//==================================================================================================
//							Beckhoff Automation Poland
//									18.04.2018
//	Struktura zawierajaca I/O odpowiedniego bloku
//  v1.0	|| TC v 3.1.4022.16		|| - pierwsza wersja
//==================================================================================================
TYPE ST_MCPowerIO:
STRUCT
	bEnable							: BOOL;
	bEnable_Positive				: BOOL;
	bEnable_Negative				: BOOL;
	lrOverride						: LREAL := 100.0;
	eBufferMode						: Tc2_MC2.MC_BufferMode;
	stOptions						: Tc2_MC2.ST_PowerOptions;
	bStatus							: bool; // Same meaning as Done
	bBusy							: BOOL;
	bActive							: BOOL;
	bError							: BOOL;
	udiErrorID						: UDINT;
END_STRUCT
END_TYPE

(* stored: Version 1.1.0.1, ProductVersion 3.1.4026.13, FileIdentifier 2b62fc5234dd54785e8d8bc13f7af48afa9d2e37, FileSignature 0c8889d59edc92878bc80d093e1a9bfaae3547ece22efeff410bd27fe71626e3a2296c260e5174e1e9f4c3579bdeef73796d740daa9c9e3fe2d72999d99b64c6bbbed3f09a929075c90ea5f568e44ca7fe1e50993d392086edb34f059cab27661d17cb18b777a1cc143007599acff074534794e17a4e454b3f07a7351b07a428d507a2aea050cb1244c9295b3d2963c55e13be54645ee29099e6efd735831ae0088fdcc0c097de074772bbfef655b8e8e41d1a06ae80c8213d93fc8d008c4355bb2c6775e5eeb260032a921d3824f40b037280879efc002fea0ec84b400487ace8bd4238f26cf557ce1b3c3b1019d7537b98cfe399dec65fd8fb329882550153
   DUT ST_MCPowerIO: Id {e4a69ddf-609c-434d-b90f-f11f6aa8257c} *)
